SYSTEM separatedAlphabot
  (* Version 1.0, 2023-01-19, test *)
  APPLICATION separatedAlphabot
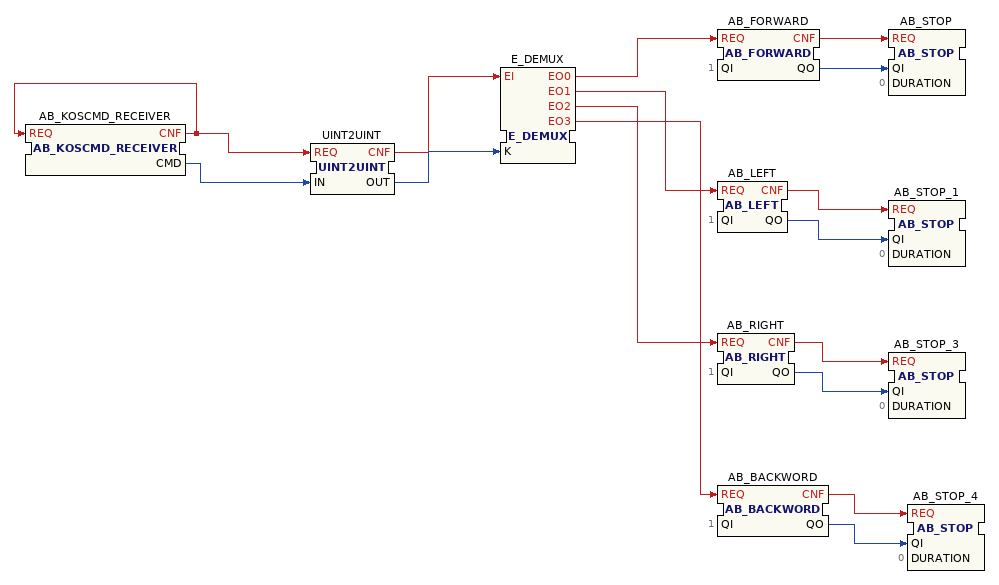
    FBS
      AB_BACKWORD : AB_BACKWORD(QI := 1);
      AB_FORWARD : AB_FORWARD(QI := 1);
      AB_STOP : AB_STOP(DURATION := 0);
      E_DEMUX : E_DEMUX;
      AB_LEFT : AB_LEFT(QI := 1);
      AB_RIGHT : AB_RIGHT(QI := 1);
      AB_STOP_1 : AB_STOP(DURATION := 0);
      AB_STOP_3 : AB_STOP(DURATION := 0);
      AB_STOP_4 : AB_STOP(DURATION := 0);
      AB_KOSCMD_RECEIVER : AB_KOSCMD_RECEIVER;
      UINT2UINT : UINT2UINT;
    END_FBS
    EVENT_CONNECTIONS
      AB_FORWARD.CNF TO AB_STOP.REQ;
      E_DEMUX.EO0 TO AB_FORWARD.REQ;
      E_DEMUX.EO1 TO AB_LEFT.REQ;
      E_DEMUX.EO2 TO AB_RIGHT.REQ;
      AB_BACKWORD.CNF TO AB_STOP_4.REQ;
      AB_RIGHT.CNF TO AB_STOP_3.REQ;
      AB_LEFT.CNF TO AB_STOP_1.REQ;
      E_DEMUX.EO3 TO AB_BACKWORD.REQ;
      AB_KOSCMD_RECEIVER.CNF TO UINT2UINT.REQ;
      UINT2UINT.CNF TO E_DEMUX.EI;
      AB_KOSCMD_RECEIVER.CNF TO AB_KOSCMD_RECEIVER.REQ;
    END_CONNECTIONS
    DATA_CONNECTIONS
      AB_FORWARD.QO TO AB_STOP.QI;
      AB_BACKWORD.QO TO AB_STOP_4.QI;
      AB_RIGHT.QO TO AB_STOP_3.QI;
      AB_LEFT.QO TO AB_STOP_1.QI;
      AB_KOSCMD_RECEIVER.CMD TO UINT2UINT.IN;
      UINT2UINT.OUT TO E_DEMUX.K;
    END_CONNECTIONS
  END_APPLICATION
  DEVICE FORTE_PC : FORTE_PC(MGR_ID := "localhost:61499")
    {SET_ATTRIBUTE(Profile, HOLOBLOC)} (* device profile *)
    RESOURCE EMB_RES : EMB_RES
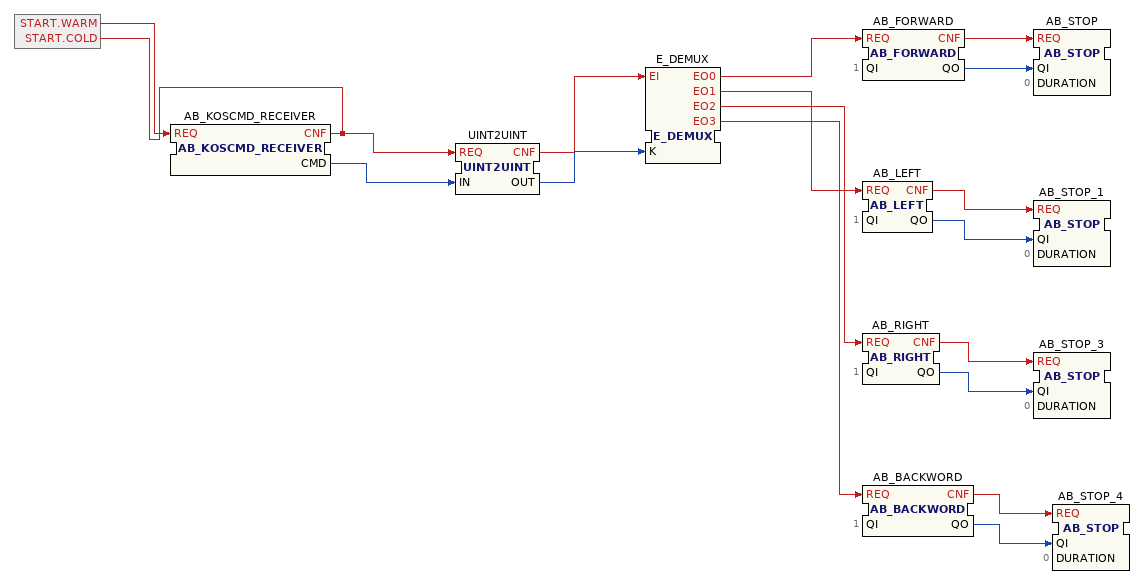
      FBS
        E_DEMUX : E_DEMUX;
        AB_FORWARD : AB_FORWARD(QI := 1);
        AB_STOP : AB_STOP(DURATION := 0);
        AB_LEFT : AB_LEFT(QI := 1);
        AB_STOP_1 : AB_STOP(DURATION := 0);
        AB_RIGHT : AB_RIGHT(QI := 1);
        AB_STOP_3 : AB_STOP(DURATION := 0);
        AB_BACKWORD : AB_BACKWORD(QI := 1);
        AB_STOP_4 : AB_STOP(DURATION := 0);
        UINT2UINT : UINT2UINT;
        AB_KOSCMD_RECEIVER : AB_KOSCMD_RECEIVER;
      END_FBS
      EVENT_CONNECTIONS
        E_DEMUX.EO0 TO AB_FORWARD.REQ;
        AB_FORWARD.CNF TO AB_STOP.REQ;
        E_DEMUX.EO1 TO AB_LEFT.REQ;
        AB_LEFT.CNF TO AB_STOP_1.REQ;
        E_DEMUX.EO2 TO AB_RIGHT.REQ;
        AB_RIGHT.CNF TO AB_STOP_3.REQ;
        E_DEMUX.EO3 TO AB_BACKWORD.REQ;
        AB_BACKWORD.CNF TO AB_STOP_4.REQ;
        UINT2UINT.CNF TO E_DEMUX.EI;
        AB_KOSCMD_RECEIVER.CNF TO AB_KOSCMD_RECEIVER.REQ;
        AB_KOSCMD_RECEIVER.CNF TO UINT2UINT.REQ;
        START.WARM TO AB_KOSCMD_RECEIVER.REQ;
        START.COLD TO AB_KOSCMD_RECEIVER.REQ;
      END_CONNECTIONS
      DATA_CONNECTIONS
        AB_FORWARD.QO TO AB_STOP.QI;
        AB_LEFT.QO TO AB_STOP_1.QI;
        AB_RIGHT.QO TO AB_STOP_3.QI;
        AB_BACKWORD.QO TO AB_STOP_4.QI;
        UINT2UINT.OUT TO E_DEMUX.K;
        AB_KOSCMD_RECEIVER.CMD TO UINT2UINT.IN;
      END_CONNECTIONS
    END_RESOURCE
  END_DEVICE
  MAPPINGS
    separatedAlphabot.E_DEMUX ON FORTE_PC.EMB_RES.E_DEMUX;
    separatedAlphabot.AB_FORWARD ON FORTE_PC.EMB_RES.AB_FORWARD;
    separatedAlphabot.AB_STOP ON FORTE_PC.EMB_RES.AB_STOP;
    separatedAlphabot.AB_LEFT ON FORTE_PC.EMB_RES.AB_LEFT;
    separatedAlphabot.AB_STOP_1 ON FORTE_PC.EMB_RES.AB_STOP_1;
    separatedAlphabot.AB_RIGHT ON FORTE_PC.EMB_RES.AB_RIGHT;
    separatedAlphabot.AB_STOP_3 ON FORTE_PC.EMB_RES.AB_STOP_3;
    separatedAlphabot.AB_BACKWORD ON FORTE_PC.EMB_RES.AB_BACKWORD;
    separatedAlphabot.AB_STOP_4 ON FORTE_PC.EMB_RES.AB_STOP_4;
    separatedAlphabot.UINT2UINT ON FORTE_PC.EMB_RES.UINT2UINT;
    separatedAlphabot.AB_KOSCMD_RECEIVER ON FORTE_PC.EMB_RES.AB_KOSCMD_RECEIVER;
  END_MAPPINGS
  SEGMENTS
    Ethernet : Ethernet;
  END_SEGMENTS
  LINKS
    FORTE_PC => Ethernet;
  END_LINKS
END_SYSTEM
